// TIA Portal project "Schleifmaschine" (V14)

(* hardware
DEVICE "S7-1200-Station_1"  S7-1200 Station
   slot 0: "Baugruppenträger_0"  S7-1200 Rack  Rack  V1.0
   slot 1: "PLC_1"  CPU 1214C DC/DC/DC  6ES7 214-1AG40-0XB0  V4.2
   slot 3: "AQ 1x12BIT_1"  AQ1 signal board  6ES7 232-4HA30-0XB0  V1.0
*)

// ===== PLC "PLC_1"  CPU 1214C DC/DC/DC =====

VAR_GLOBAL   // PLC tag table "Standard-Variablentabelle"
   "System_Byte" AT %MB100 : Byte;
   "FirstScan" AT %M100.0 : Bool;
   "DiagStatusUpdate" AT %M100.1 : Bool;
   "AlwaysTRUE" AT %M100.2 : Bool;
   "AlwaysFALSE" AT %M100.3 : Bool;
   "Clock_Byte" AT %MB110 : Byte;
   "Clock_10Hz" AT %M110.0 : Bool;
   "Clock_5Hz" AT %M110.1 : Bool;
   "Clock_2.5Hz" AT %M110.2 : Bool;
   "Clock_2Hz" AT %M110.3 : Bool;
   "Clock_1.25Hz" AT %M110.4 : Bool;
   "Clock_1Hz" AT %M110.5 : Bool;
   "Clock_0.625Hz" AT %M110.6 : Bool;
   "Clock_0.5Hz" AT %M110.7 : Bool;
   "S2" AT %I0.0 : Bool;   // Taster ( 0 ) - Öffner
   "S1" AT %I0.1 : Bool;   // Taster ( 1 ) - Schließer
   "S4" AT %I0.3 : Bool;   // Taster ( I ) - Schliesser
   "S3" AT %I0.2 : Bool;   // Taster ( STOP ) - Öffner
   "S6" AT %I0.4 : Bool;   // Taster ( II ) - Schliesser
   "S5" AT %I0.6 : Bool;   // Taster ( ← ) - Schliesser
   "S8" AT %I0.5 : Bool;   // Taster ( STOP ) - Öffner
   "S7" AT %I0.7 : Bool;   // Taster ( → ) - Schliesser
   "S10" AT %I1.1 : Bool;   // Not-Halt - Öffner
   "S11" AT %I1.0 : Bool;   // Not-Halt - Schliesser
   "Q1" AT %Q0.0 : Bool;   // Motor schnell (RL)
   "Q2" AT %Q0.1 : Bool;   // Motor Linkslauf
   "Q3" AT %Q0.2 : Bool;   // Motor langsam (RL)
   "P1" AT %Q0.4 : Bool;   // Meldeleuchte weiß
   "P2" AT %Q0.5 : Bool;   // Meldeleuchte grün
   "P3" AT %Q0.6 : Bool;   // Meldeleuchte rot
   "AlleAusgänge" AT %QW0 : Word;
END_VAR

FUNCTION "fc_Getriebemotor" : Void   // FC1, FBD
{ S7_Optimized_Access := 'TRUE' }
VERSION : 0.1
BEGIN

REGION Network 1: Motor schnell (RL)
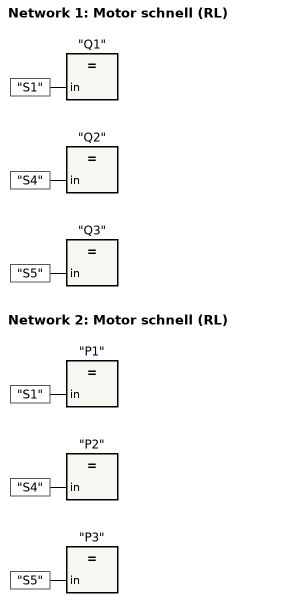
   "Q1" := "S1";
   "Q2" := "S4";
   "Q3" := "S5";
END_REGION

REGION Network 2: Motor schnell (RL)
   "P1" := "S1";
   "P2" := "S4";
   "P3" := "S5";
END_REGION
END_FUNCTION

ORGANIZATION_BLOCK "Main"   // OB1, LAD, ProgramCycle
TITLE = "Main Program Sweep (Cycle)"
{ S7_Optimized_Access := 'TRUE' }
VERSION : 0.1
   VAR_INPUT
      Initial_Call : Bool;   // Initial call of this OB
      Remanence : Bool;   // =True, if remanent data are available
   END_VAR
BEGIN

REGION Network 1
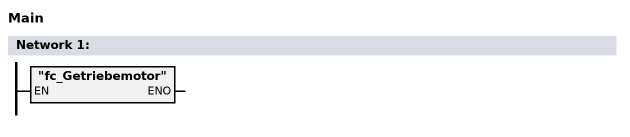
   RUNG wire#powerrail
      "fc_Getriebemotor"()
   END_RUNG
   // the same network as SCL:
   "fc_Getriebemotor"();
END_REGION
END_ORGANIZATION_BLOCK

ORGANIZATION_BLOCK "Startup"   // OB100, SCL, Startup
TITLE = "Complete Restart"
{ S7_Optimized_Access := 'TRUE' }
VERSION : 0.1
   VAR_INPUT
      LostRetentive : Bool;   // True if retentive data are lost
      LostRTC : Bool;   // True if date and time are lost
   END_VAR
BEGIN
   "AlleAusgänge" := 16#0000;
END_ORGANIZATION_BLOCK